// TwinCAT 3 PLC project SPS
// Company: mbc engineering GmbH
// ProgramVersion: 3.1.4022.2
// libraries:
//   Tc2_Standard, * (Beckhoff Automation GmbH)
//   Tc2_System, * (Beckhoff Automation GmbH)
//   Tc3_Module, * (Beckhoff Automation GmbH)
//   MBC TC3 PCS Library,newest,mbc engineering GmbH
// project tree:
//   Commands/ AddCommand.TcPOU (not stored), Commands.TcGVL, DelayedAddCommand.TcPOU (not stored), PRG_Commands.TcPOU, StartCommand.TcPOU
//   / PlcTask.TcTTO (not stored)
//   POUs/ MAIN.TcPOU

// ---- Commands/Commands.TcGVL
{attribute 'qualified_only'}
VAR_GLOBAL
	StartCommand1		: StartCommand;
	AddCommand1			: AddCommand 			:= (Val1 := 3, Val2 := 2);
	DelayedAddCommand1	: DelayedAddCommand 	:= (Val1 := 4, Val2 := 5);
END_VAR

// ---- Commands/StartCommand.TcPOU
FUNCTION_BLOCK PUBLIC StartCommand EXTENDS CommandBase
VAR_INPUT
END_VAR
VAR_OUTPUT
	Q : BOOL;
END_VAR
VAR
	bInit 	: BOOL;
END_VAR

// Will be executed in the same cycle ``stHandshake.bExecute`` changes to ``true``
METHOD PROTECTED Init
bInit := TRUE;
END_METHOD

// Execute the funktional part of the command implementation. Will be executed in the same cycle ``stHandshake.bExecute`` changes to ``true`` after the ``Init`` Method
METHOD PROTECTED Task : BOOL
// Task Code:
// dedect task completed
IF (NOT bInit AND Q) THEN
	// Task comlete;
	Task := SUPER^.Task();;
END_IF

// set output trigger
Q := bInit;

// Reset after 1. cycle
bInit := FALSE;
END_METHOD

END_FUNCTION_BLOCK

// ---- Commands/PRG_Commands.TcPOU
PROGRAM PRG_Commands
VAR
	fbTofStartCommand1		: TOF;		// Shows the exection was happen
END_VAR

Commands.StartCommand1.Call();
	
fbTofStartCommand1(
	IN := Commands.StartCommand1.Q,
	PT := T#1S);	
	
	
Commands.AddCommand1.Call();
Commands.DelayedAddCommand1.Call();

END_PROGRAM

// ---- POUs/MAIN.TcPOU
PROGRAM MAIN
VAR
	counter				: UINT;
END_VAR

counter := counter + 1;

PRG_Commands();

END_PROGRAM
